PROGRAM main
VAR
	Fast_Mode_Button AT %IX0.0 : bool;
	Slow_Mode_Button AT %IX0.1 : bool;
	LED AT %QX0.0 : bool;
	Blink_Time : time;
	TON_ON : TON;
	TON_OFF : TON;
END_VAR

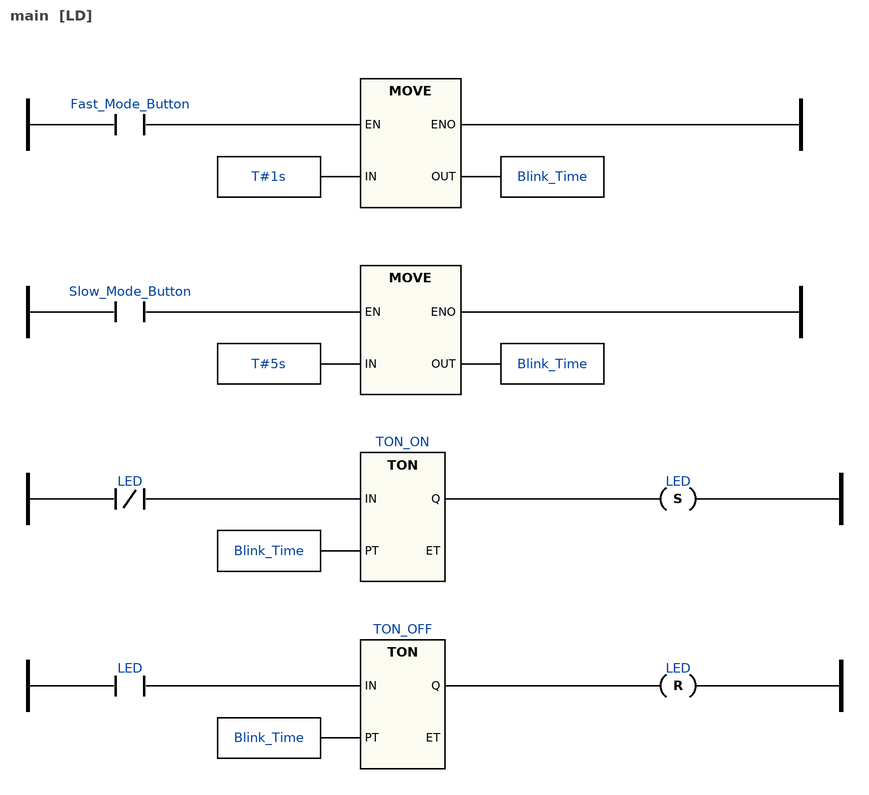
(* LD diagram, written out as Structured Text *)
IF Fast_Mode_Button THEN Blink_Time := T#1s; END_IF;
IF Slow_Mode_Button THEN Blink_Time := T#5s; END_IF;
TON_ON(IN := NOT LED, PT := Blink_Time);
IF TON_ON.Q THEN LED := TRUE; END_IF;
TON_OFF(IN := LED, PT := Blink_Time);
IF TON_OFF.Q THEN LED := FALSE; END_IF;
END_PROGRAM
